// TIA Portal V16 export
// export: Created 2024-03-27T10:00:40.3167068Z, ExportSetting WithDefaults, DisplayName Totally Integrated Automation Portal, DisplayVersion V16, DisplayName TIA Portal Version Control Interface, DisplayVersion V16, DisplayName TIA Portal Openness, DisplayVersion V16, DisplayName STEP 7 Professional, DisplayVersion V16, DisplayName STEP 7 Safety, DisplayVersion V16, DisplayName WinCC Advanced, DisplayVersion V16
DATA_BLOCK "AssemblageCel_U_DB"   // DB1
VERSION : 0.1
// stored: AutoNumber true, DBAccessibleFromOPCUA true, InstanceOfName AssemblageCel_U, InstanceOfType FB
"AssemblageCel_U"
   // VAR_INPUT
   //    Start : Bool;
   //    Stop : Bool;
   //    EStop : Bool;
   // END_VAR
   // VAR
   //    Stap : Int;
   //    Prev_Stap : Int;
   //    Lagerpers : "Lagerpers_EM";
   //    Draaitafel { S7_SetPoint := 'True'} : "Draaitafel_EM";
   //    Cobot { S7_SetPoint := 'True'} : "Cobot_EM";
   // END_VAR
BEGIN
END_DATA_BLOCK
